PROGRAM FbdRule
VAR
END_VAR

// NETWORK 1

END_PROGRAM

(* stored: Version 1.1.0.1, ProductVersion 3.1.4024.12
   POU FbdRule: Id {9ad0727c-58a9-47e5-885c-9b7c1f73be00}, SpecialFunc None *)
